(* PLC project Generated.project, CODESYS CODESYS V3.5 SP19 Patch 1 *)
(* stored: creationDateTime 2026-11-18T13:32:59.811305, modificationDateTime 2026-11-18T13:32:59.811305 *)

(* values of E_MachineHomingStep: IDLE: Referencement indisponible (Enable=FALSE); LOSS_SAFESTOP: Perte de datum en mouvement : arret controle en cours; BOTH_NOT_HOMED: Codeurs M1 et M2 non references : passer en MAINT_N2; M1_NOT_HOMED: Codeur M1 non reference ou mesure douteuse : homer M1; M2_NOT_HOMED: Codeur M2 non reference ou mesure douteuse : homer M2; OFFSET_UNKNOWN: Offset benne inconnu : passer en MAINT_N2; NEED_TOP_POSITION: Monter Both a vitesse lente jusqu au capteur haut; NEED_MECHANICAL_STOP: Capteur haut atteint : relacher la commande et attendre l arret; AWAIT_BUCKET_CONFIRM: Confirmer visuellement la benne : Fermee ou Ouverte; HOMING_IN_PROGRESS: Referencement conjoint M1/M2 en cours : ne pas manoeuvrer; VALID: Referencement machine valide : mode nominal disponible; FAILED: Referencement incomplet : rester en N2 et recommencer *)

{attribute 'qualified_only'}
{attribute 'strict'}
TYPE E_MachineHomingStep : (IDLE := 0, LOSS_SAFESTOP := 5, BOTH_NOT_HOMED := 10, M1_NOT_HOMED := 11, M2_NOT_HOMED := 12, OFFSET_UNKNOWN := 20, NEED_TOP_POSITION := 30, NEED_MECHANICAL_STOP := 40, AWAIT_BUCKET_CONFIRM := 45, HOMING_IN_PROGRESS := 50, VALID := 60, FAILED := 70);
END_TYPE

(* values of E_MachineHomingTxState: HX0_REPOS: Repos : N1 libre bloque si NOT Homed, M3 bloque N1/SEMI, attente 5s BP joy N1 ou BtnStart N2; HX1_BUCKET_PREPARE: M2 seul palier 1, ouv + ferm sans butees soft, garde continue 20s + decompte, BtnValidate neutre; HX2_CLIMB_TO_TOP: Couple M1+M2 palier 1 : montee lente + detente 2s max/geste, viser avant TOP sans toucher; HX3_TOP_CLEARANCE: Contact TOP = perdu/surcourse -> montee interdite, descente ~4s apres relachement TOP -> retour HX1; HX4_FINAL_CONFIRM: Arret avant TOP + avertissement -> BtnValidate neutre -> preset 8.5m M1+M2 + CommitClose -> Homed; HX7_FAILED: Echec / abandon : coupure mouvements, purge etats, attente Reset conscient *)

{attribute 'qualified_only'}
{attribute 'strict'}
TYPE E_MachineHomingTxState : (HX0_REPOS := 0, HX1_BUCKET_PREPARE := 1, HX2_CLIMB_TO_TOP := 2, HX3_TOP_CLEARANCE := 3, HX4_FINAL_CONFIRM := 4, HX7_FAILED := 5);
END_TYPE

(* values of E_Mode: DISABLE: Mode Désactivé / Veille de sécurité (sorties bloquées); MAINT_N1: Manuel Niveau 1 : Pilotage unitaire avec toutes sécurités actives; MAINT_N2: Manuel Niveau 2 : Pilotage dégradé (droits étendus + bypasses autorisés); SEMI_AUTO: Mode Semi-Automatique (séquenceur automatique) *)

{attribute 'qualified_only'}
{attribute 'strict'}
TYPE E_Mode : (DISABLE := 0, MAINT_N1 := 1, MAINT_N2 := 2, SEMI_AUTO := 3);
END_TYPE

(* ======================================================================= 🧩 ST_Fault — Brique socle défaut (2 vues : live + latchée) ─────────────────────────────────────────────────────────────── 🎯 Rôle : porter l'état défaut d'un composant, applicable dans TOUS les cas (acquittable ou non), sans brique warning séparée. • Vue LIVE (Error / ErrorId) : suit la cause, retombe seule à 0. • Vue LATCHÉE (Latched / LatchedId): mémorisée au défaut, reste jusqu'au front Reset. Le choix acquittable / non-acquittable se fait PAR CAUSE (ST_FaultCause.Latching), jamais par bloc. 🔒 Sécurité : interlock TOUJOURS sur la cause brute (Error / ErrorId), jamais sur l'acquittement. Reset TOUJOURS effectif, jamais conditionné (std §9). 🧬 Composition : brique de base réutilisable — sortie de FB, struct métier, GVL. Texte IHM NON stocké ici : dérivé côté IHM depuis LatchedId / ErrorId. 📄 Doc : DOC/STDS/CODE_QUALITY_STANDARDS.md §2quinquies / §9 ======================================================================= *)
TYPE ST_Fault : STRUCT
  Error : BOOL;  (* <-- [DIAG] vue LIVE : au moins une cause présente maintenant *)
  ErrorId : WORD;  (* <-- [DIAG] bitfield des causes présentes maintenant (0 si aucune) *)
  Latched : BOOL;  (* <-- [DIAG] vue LATCHÉE : défaut non acquitté, reste jusqu'au front Reset *)
  LatchedId : WORD;  (* <-- [DIAG] ErrorId figé à l'apparition du défaut, effacé au Reset *)
END_STRUCT;
END_TYPE

(* ======================================================================= 🧩 ST_FaultCause — Cause élémentaire alimentant ST_Fault (socle FB_FaultCore) ─────────────────────────────────────────────────────────────── 🎯 Rôle : une cause exprimée EN CLAIR (BOOL + libellé), sans bitfield ni masque. Le FB métier remplit une liste (ARRAY[0..15] OF ST_FaultCause) ; le socle FB_FaultCore en déduit ST_Fault (vue live + vue latchée). 🔒 Sécurité : interlock TOUJOURS sur Active (cause brute), jamais sur le latch. Latching = TRUE → la cause ARME la vue latchée (défaut à acquitter). Latching = FALSE → la cause n'alimente que la vue live (retombe seule). Fail-safe : une cause laissée à Latching=FALSE reste visible en live — pour la rendre acquittable, il faut le déclarer explicitement. 📄 Doc : DOC/STDS/CODE_QUALITY_STANDARDS.md §2quinquies / §9 ======================================================================= *)
TYPE ST_FaultCause : STRUCT
  Active : BOOL;  (* 1 = cause présente maintenant (interlock sur cette valeur) *)
  Latching : BOOL;  (* 1 = cause à acquitter (arme Latched) ; 0 = live seulement *)
  Texte : STRING;  (* libellé prêt IHM (non stocké dans ST_Fault, dérivé côté IHM) *)
END_STRUCT;
END_TYPE

(* ======================================================================= 🧩 ST_Lifecycle — Brique socle cycle d'exécution ─────────────────────────────────────────────────────────────── 🎯 Rôle : porter l'avancement d'une action à cycle (organe, séquenceur). Optionnelle : un FB purement synchrone (conditionneur, filtre, joystick) ne la porte pas. 🧬 Composition : brique de base réutilisable, composée avec ST_Fault. 📄 Doc : DOC/STDS/CODE_QUALITY_STANDARDS.md §2quinquies ======================================================================= *)
TYPE ST_Lifecycle : STRUCT
  Busy : BOOL;  (* <-- [STAT] 1 = action en cours *)
  Done : BOOL;  (* <-- [STAT] 1 = action terminée avec succès *)
END_STRUCT;
END_TYPE

(* ======================================================================= 🔌 ST_ProgramWinchRequest — Demande de mouvement treuil par le programme ─────────────────────────────────────────────────────────────── 🎯 Rôle : Regroupe les demandes logiques de treuil formulées par le séquenceur 📄 Référentiel : DOC/WFLOW/CONTRACTS/INTERPRG_CONTRACT_PRG03_MODES_CYCLE_v1.0.md ======================================================================= *)
TYPE ST_ProgramWinchRequest : STRUCT
  RunRequest : BOOL;  (* Ordre marche demandé par le programme *)
  ReqAscent : BOOL;  (* Demande montée *)
  ReqDescend : BOOL;  (* Demande descente *)
  StepTgt : INT;  (* Palier de vitesse cible demandé (1 à 5, 0 = arrêt) *)
END_STRUCT;
END_TYPE

(* ======================================================================= 🔌 ST_fbMachineHomingCycle_AxisHomingStatus — Statut homing d'un axe treuil ─────────────────────────────────────────────────────────────── 🎯 Rôle : Regroupe l'etat de homing d'un axe (M1 ou M2) consomme par FB_CycleMachineHoming pour piloter le guide et la transaction. 📄 Doc métier : DOC/AF/AF_Partie-09_Fonction_Encoder_v2.4.md (F09.08) ======================================================================= *)
TYPE ST_fbMachineHomingCycle_AxisHomingStatus : STRUCT
  HomedAndReliable : BOOL;  (* Codeur reference ET mesure jugee fiable (gate strict) *)
  HomingBusy : BOOL;  (* Sequence de homing en cours sur l'axe *)
  HomingDone : BOOL;  (* Homing termine avec succes (HomingLifecycle.Done cote FB_Encoder) *)
  HomingError : BOOL;  (* Homing en erreur sur l'axe (HomingFault.Error) *)
  HomingProvisional : BOOL;  (* TRUE si le datum persistant RETAIN est provisoire (HX1 0m) *)
END_STRUCT;
END_TYPE

(* ======================================================================= 🔌 ST_fbMachineHomingCycle_BucketCommit — Commit atomique de l'etat benne ─────────────────────────────────────────────────────────────── 🎯 Rôle : Impulsion 1 scan emise par FB_CycleMachineHoming vers FB_Bucket apres succes des DEUX homings. FB_Bucket reste seul proprietaire de IsOpen / IsClosed. 🔒 Sécurité : CommitOpen et CommitClose mutuellement exclusifs (garanti par le corps du FB — rejet du double-confirm, cf. C-2). 📄 Doc métier : DOC/AF/AF_Partie-05_Modes_Maintenance_v2.1.md ======================================================================= *)
TYPE ST_fbMachineHomingCycle_BucketCommit : STRUCT
  CommitOpen : BOOL;  (* Publier "benne ouverte" (impulsion 1 scan) *)
  CommitClose : BOOL;  (* Publier "benne fermee" (impulsion 1 scan) *)
  CommitInvalidate : BOOL;  (* Revoquer reference benne (abandon avant calibration altimetrie) *)
END_STRUCT;
END_TYPE

(* ======================================================================= ⚙️ ST_fbMachineHomingCycle_Cfg — Réglages de FB_CycleMachineHoming ─────────────────────────────────────────────────────────────────────── 🎯 Rôle : Réglages géométriques du référencement machine (cible haute M2/benne + écarts benne) + temporisations de garde du GRAFCET de homing (montée, homing axes). 🔒 Ownership : produit par PRG_02_Acquisition depuis _WinchM2CfgPersist (cible haute) et _BucketCfgPersist (écarts, GVL_PERSISTENT). Initialized : drapeau de restauration boot (pont persistant). 📄 Doc métier : DOC/AF/AF_Partie-09_Fonction_Encoder_v2.4.md (F09.08) ======================================================================= *)
TYPE ST_fbMachineHomingCycle_Cfg : STRUCT
  CfgTopHomingTarget_M : REAL;  (* Position capteur haut M2/benne (m) — cible finale HX4 M2 (+ OffsetCloseM) *)
  CfgTopHomingTargetM1_M : REAL := 8.5;  (* Position capteur haut M1 (m) — cible finale HX4 M1 (defaut 8.5 m) *)
  CfgOffsetOpen_M : REAL;  (* Ecart géométrique benne ouverte (m) *)
  CfgOffsetClose_M : REAL;  (* Ecart géométrique benne fermée (m) *)
  CfgTimeoutClimb : TIME := TIME#300s0ms;  (* Garde de montee : budget d'une MONTER CONTINUE (un temporisateur remet son temps ecoule a zero des que la commande retombe : une pause operateur ou un arret d'urgence ne consomme donc rien). Derivation : course maximale de cable = CfgTopSensorPos_M - CfgCableLimitDescent_M (8,5 m - (-50 m) = 58,5 m) ; borne haute de vitesse du palier 1 = 0,4 m/s (GVL_PERSISTENT._WinchSpeedConfig.SpeedBandMaxMps[1], valeur de banc A MESURER sur site) => 58,5 / 0,4 = 146,3 s ; marge x2 = 292,5 s ; valeur retenue 300 s (arrondie au-dessus). A revoir si la course ou la vitesse du palier 1 changent (gate G511). Garde de montee au capteur haut (0 = pas de garde) *)
  CfgEntryHoldTime : TIME := TIME#5s0ms;  (* Duree maintien BP joystick au neutre en HX0 (MAINT_N1) *)
  CfgBucketPrepareTimeout : TIME := TIME#20s0ms;  (* Duree max commande continue M2 en HX1 (coupe -> neutre) *)
  CfgSlackReliefMaxTime : TIME := TIME#2s0ms;  (* Duree max descente detente cable par geste en HX2 *)
  CfgTopClearanceTime : TIME := TIME#4s0ms;  (* Duree descente accumulee apres relachement TOP en HX3 *)
  CfgTimeoutHomeAxes : TIME := TIME#60s0ms;  (* Garde globale prise de reference (HX4) *)
  Initialized : BOOL := FALSE;  (* Drapeau de restauration config au boot (pont persistant) *)
END_STRUCT;
END_TYPE

(* ======================================================================= 🔌 ST_fbMachineHomingCycle_HomingDemand — Demande de homing conjoint vers un axe ─────────────────────────────────────────────────────────────── 🎯 Rôle : Ordre de prise d'origine emis par FB_CycleMachineHoming vers une facade FB_Encoder. M1 : cible configuree. M2 : cible geometrique dynamique (top M1 configure +/- offset benne), jamais une position M1 live. 📄 Doc métier : DOC/AF/AF_Partie-09_Fonction_Encoder_v2.4.md (F09.08) ======================================================================= *)
TYPE ST_fbMachineHomingCycle_HomingDemand : STRUCT
  HomeReq : BOOL;  (* Demande de prise d'origine pour cet axe (vocab reserve Homing) *)
  UseDynamicTarget : BOOL;  (* TRUE => cible = DynamicTarget_M (M2 uniquement) *)
  DynamicTarget_M : REAL;  (* Cible geometrique benne (m) : CfgTopHomingTargetM + offset *)
  Provisional : BOOL;  (* TRUE => marque Calib.HomingProvisional RETAIN (zero provisoire HX1) *)
END_STRUCT;
END_TYPE

(* ======================================================================= 🎯 FB_CycleMachineHoming — Cycle de referencement machine M1/M2/benne ─────────────────────────────────────────────────────────────── Role : GRAFCET sequentiel 5 etapes (HX0..HX4 + HX7_FAILED) : - HX0_REPOS : N1 libre bloque si NOT Homed, M3 verrouille N1/SEMI (echappatoire N2), entree par 5s BP joystick au neutre (N1) ou BtnStart (N2). Jamais relanceable si MachineHomed = TRUE. - HX1_BUCKET_PREPARE : M2 seul palier 1, ouv + ferm sans butees soft, garde continue 20s + decompte message, BtnValidate neutre. - HX2_CLIMB_TO_TOP : Couple M1+M2 palier 1, montee lente + detente cable max 2s par geste, viser avant TOP sans le toucher. - HX3_TOP_CLEARANCE : Contact TOP = surcourse/perdu -> coupure montee, descente ~4s accumulee apres relachement TOP -> retour HX1. - HX4_FINAL_CONFIRM : Arret avant TOP + avertissement + BtnValidate neutre -> preset 8.5m M1 + (8.5m + OffsetCloseM) M2 + CommitClose. Doc metier : DOC/WFLOW/MISE_EN_SERVICE/PLAN_REFONTE_GRAFCET_HOMING_20261118_v1.0.md + DOC/AF/AF_Partie-09_Fonction_Encoder_v2.4.md (F09.08) ======================================================================= *)
FUNCTION_BLOCK FB_CycleMachineHoming
  VAR_INPUT
    Enable : BOOL;  (* === CONTRAT STANDARD (Enable + Reset) === --> [CMD] Autorisation generale *)
    Reset : BOOL;  (* --> [CMD] Acquittement defaut / abandon cycle (front) *)
    Mode : E_Mode;  (* === MODE ARBITRE === --> [CMD] Mode machine (MAINT_N1 ou MAINT_N2 autorises) *)
    BootReady : BOOL;  (* --> [HW] Acquisition + codeurs valides apres boot *)
    TopPositionSensor : BOOL;  (* === PERMIS SECURITE === --> [SAFE] Capteur haut commun M1/M2 (TRUE = atteint) *)
    TopHardStopLatched : BOOL := FALSE;  (* --> [SAFE] Latch directionnel capteur haut (PRG_06_Outputs) *)
    WinchesMechanicallyStopped : BOOL;  (* --> [SAFE] M1 ET M2 arret mecanique confirme *)
    BucketIsOpen : BOOL := FALSE;  (* --> [HW] Benne ouverte confirmee (PRG_04_Treuils_Benne) *)
    M1Status : ST_fbMachineHomingCycle_AxisHomingStatus;  (* === ACQUISITION HOMING (M1 / M2) === --> [HW] Statut homing axe M1 *)
    M2Status : ST_fbMachineHomingCycle_AxisHomingStatus;  (* --> [HW] Statut homing axe M2 *)
    BucketOffsetValid : BOOL;  (* === ETAT BENNE === --> [HW] Reference benne persistante valide *)
    DeadmanArmed : BOOL;  (* === PERMIS OPERATEUR (joystick + homme-mort) === --> [CMD] Homme-mort arme *)
    RawDeadmanButton : BOOL := FALSE;  (* --> [HW] BP joystick brut (sert en HX0 N1 quand ArmingPermit=FALSE) *)
    JoystickDeflected : BOOL;  (* --> [CMD] Joystick deflechi (X ou Y hors neutre) *)
    JoystickPull : BOOL;  (* --> [CMD] Manche tire = montee / fermeture benne *)
    JoystickPush : BOOL;  (* --> [CMD] Manche pousse = descente / ouverture benne *)
    BtnValidation : BOOL;  (* === VALIDATION OPERATEUR === --> [CMD] Bouton validation IHM unifie (HX1, HX2->HX4, HX4) *)
    StartRequest : BOOL;  (* --> [CMD] Bouton Start IHM (HX0 en MAINT_N2) *)
    BtnConfirmHomingBucket : BOOL;  (* --> [CMD] Compat bouton IHM historique HX1 *)
    JoystickWinchSelectArbitrated : INT;  (* === INTERLOCK COUPLAGE E1 & RETOUR ARBITRAGE === --> [CMD] Selecteur treuil arbitre aval (0=couple, 2=M2) *)
    CablePosM1 : REAL;  (* === MESURES POSITIONS === --> [MEAS] Position cable M1 (m) *)
    CablePosM2 : REAL;  (* --> [MEAS] Position cable M2 (m) *)
    CoherenceLimitM : REAL := 1;  (* --> [CFG] Coherence (compat) *)
    CfgCommissioningEnable : BOOL;  (* === MISE EN SERVICE : forcage de step (encadre) === --> [CFG] Case mise en service *)
    CfgForceStepTarget : INT;  (* --> [CFG] Step cible [0..5] *)
    CfgForceStepApply : BOOL;  (* --> [CMD] Front d'application forcage *)
    Cfg : ST_fbMachineHomingCycle_Cfg;  (* === REGLAGES & CONFIGURATION === --> [CFG] Reglages + temporisations *)
  END_VAR
  VAR_OUTPUT
    Ready : BOOL;  (* === CONTRAT STANDARD === *)
    Fault : ST_Fault;
    Lifecycle : ST_Lifecycle;
    MachineHomed : BOOL;  (* === QUALIFICATION MACHINE === *)
    MachineHomingStep : E_MachineHomingStep := E_MachineHomingStep.IDLE;
    MachineHomingStepAtError : E_MachineHomingStep := E_MachineHomingStep.IDLE;
    MachineHomingSeqStep : E_MachineHomingTxState := E_MachineHomingTxState.HX0_REPOS;
    MachineHomingInstruction : STRING(120);
    MachineHomingActionText : STRING(120);
    MachineHomingActive : BOOL;
    MachineHomingLossSafeStop : BOOL;
    MachineHomingFailed : BOOL;
    HomingModeBActive : BOOL;
    M1Demand : ST_fbMachineHomingCycle_HomingDemand;  (* === DEMANDES HOMING (M1 / M2) === *)
    M2Demand : ST_fbMachineHomingCycle_HomingDemand;
    CmdWinchM1 : ST_ProgramWinchRequest;  (* === ORDRES / PERMIS VERS PRG_03 / PRG_04 === *)
    CmdWinchM2 : ST_ProgramWinchRequest;
    CmdBucketOpen : BOOL;
    CmdBucketClose : BOOL;
    CmdWinchSelect : INT := -1;
    AllowAscent : BOOL;
    AllowDescend : BOOL;
    SoftLimitsOff : BOOL;
    InvalidateProvisionalDatum : BOOL;
    BucketCommit : ST_fbMachineHomingCycle_BucketCommit;  (* === COMMIT BENNE === *)
    M3Locked : BOOL;  (* === VERROU TRANSLATION === *)
    TopContactLatched : BOOL;  (* === LATCH & COMPTEUR CONTACT TOP HOMING === *)
    TopContactCount : UINT;
  END_VAR
  VAR
    instFault : FB_FaultCore;  (* === SOUS-INSTANCES === *)
    ResetEdge : R_TRIG;
    LatchedEdge : R_TRIG;
    StartEdge : R_TRIG;
    BtnValidationEdge : R_TRIG;
    HomingBucketConfirmEdge : R_TRIG;
    ForceStepApplyEdge : R_TRIG;
    instCauses : ARRAY[0..15] OF ST_FaultCause;
    SeqStep : E_MachineHomingTxState := E_MachineHomingTxState.HX0_REPOS;  (* === GRAFCET & ETATS INTERNES === *)
    CommitPublished : BOOL;
    CycleRunning : BOOL;
    FirstScanDone : BOOL;
    RawBtnSeenReleased : BOOL;
    Step1MoveCutoff : BOOL;
    Step1PresetIssued : BOOL;
    Step2SlackCutoff : BOOL;
    Step3BucketOpenDone : BOOL;
    Step3ClearanceDone : BOOL;
    Step4PresetIssued : BOOL;
    Step4AutoConfirmPending : BOOL;
    ProvisionalDatumActive : BOOL;
    ProvisionalAborted : BOOL;
    ForceStepClamped : INT;
    EntryHoldTimer : TON;  (* === TEMPORISATIONS === *)
    RecoveryHoldTimer : TON;
    StepValidateHoldTimer : TON;
    Step1MoveTimer : TON;
    Step2SlackTimer : TON;
    Step3Timer : TON;
    Step3AccumTime : TIME;
    Step3SegTime : TIME;
    Step3RemainingTime : TIME;
    Step3TimerRunning : BOOL;
    ClimbTimer : TON;
    HomeAxesTimer : TON;
    CouplingSettleTimer : TON;
    CouplingViolationTimer : TON;
    SettleGraceTimer : TON;
    EntryRemSec : INT;  (* === CALCULS AFFICHAGE === *)
    RecoveryRemSec : INT;
    ValRemSec : INT;
    Step1RemSec : INT;
    Step3RemSec : INT;
    BothAxesHomed : BOOL;  (* === CONDITIONS INTERMEDIAIRES === *)
    CommitOrOffsetValid : BOOL;
    ClimbPermit : BOOL;
    TopBlockedAtEntry : BOOL;
    RecoveryCauseGone : BOOL;
    EffectiveResetPulse : BOOL;
    Step1MovingCmd : BOOL;
    Step2SlackCmd : BOOL;
    Step3DescendEngaged : BOOL;
    StepValidateAllowed : BOOL;
    StepValidateHoldActive : BOOL;
    IsInMovePhase : BOOL;
    AxisHomingError : BOOL;
    MotionOutOfPhase : BOOL;
    ModeChangedInCycle : BOOL;
    ClimbTimedOut : BOOL;
    HomeAxesTimedOut : BOOL;
    TransactionAbort : BOOL;
    ReHomingAckRequired : BOOL;
    MachineWasHomed : BOOL;
    HomingLossLatched : BOOL;
    MachineHomedRaw : BOOL;
    AxesDatumRaw : BOOL;
    PrevMode : E_Mode := E_Mode.DISABLE;  (* === CONTEXTE MODES & INTERLOCKS === *)
    ModeIsMaint1 : BOOL;
    ModeIsMaint2 : BOOL;
    MaintenanceActive : BOOL;
    ClimbStepActive : BOOL;
    ClimbCommandActive : BOOL;
    CouplingInterlockFault : BOOL;
    ValidatePressed : BOOL;
    CST_CauseHomingLostInMotion : INT := 0;
    CST_CauseClimbTimeout : INT := 1;
    CST_CauseMotionOutOfPhase : INT := 2;
    CST_CauseHomingErrorM1 : INT := 3;
    CST_CauseHomingErrorM2 : INT := 4;
    CST_CauseHomeAxesTimeout : INT := 5;
    CST_CauseCouplingFault : INT := 6;
    CST_SettleGrace : TIME := TIME#3s0ms;
  END_VAR

            

{region "§1 Fronts, remises a zero de tete de scan"}
IF NOT FirstScanDone THEN
    SeqStep              := E_MachineHomingTxState.HX0_REPOS;
    MachineHomingSeqStep := E_MachineHomingTxState.HX0_REPOS;
    MachineHomingFailed  := FALSE;
    HomingModeBActive    := FALSE;
    RawBtnSeenReleased   := NOT RawDeadmanButton;
    Step1MoveCutoff      := FALSE;
    Step1PresetIssued    := FALSE;
    Step2SlackCutoff     := FALSE;
    Step3BucketOpenDone  := FALSE;
    Step3ClearanceDone   := FALSE;
    Step3AccumTime       := T#0s;
    Step3SegTime         := T#0s;
    Step3RemainingTime   := T#0s;
    Step3TimerRunning    := FALSE;
    Step3Timer(IN := FALSE, PT := T#0s);
    EntryHoldTimer(IN := FALSE, PT := T#0s);
    RecoveryHoldTimer(IN := FALSE, PT := T#0s);
    StepValidateHoldTimer(IN := FALSE, PT := T#0s);
    Step4PresetIssued       := FALSE;
    Step4AutoConfirmPending := FALSE;
    ProvisionalDatumActive  := FALSE;
    ProvisionalAborted      := FALSE;
    TopContactLatched       := FALSE;
    TopContactCount         := 0;
    PrevMode                := Mode;
END_IF;

// Sorties impulsionnelles et permis remis a zero en tete de scan
M1Demand.HomeReq := FALSE; M1Demand.UseDynamicTarget := FALSE; M1Demand.DynamicTarget_M := 0.0; M1Demand.Provisional := FALSE;
M2Demand.HomeReq := FALSE; M2Demand.UseDynamicTarget := FALSE; M2Demand.DynamicTarget_M := 0.0; M2Demand.Provisional := FALSE;
BucketCommit.CommitOpen       := FALSE;
BucketCommit.CommitClose      := FALSE;
BucketCommit.CommitInvalidate := FALSE;
InvalidateProvisionalDatum    := FALSE;
CmdBucketOpen  := FALSE;
CmdBucketClose := FALSE;
CmdWinchM1.RunRequest := FALSE; CmdWinchM1.ReqAscent := FALSE; CmdWinchM1.ReqDescend := FALSE; CmdWinchM1.StepTgt := 0;
CmdWinchM2.RunRequest := FALSE; CmdWinchM2.ReqAscent := FALSE; CmdWinchM2.ReqDescend := FALSE; CmdWinchM2.StepTgt := 0;
CmdWinchSelect := -1;
AllowAscent    := FALSE;
AllowDescend   := FALSE;
SoftLimitsOff  := FALSE;

ResetEdge(CLK := Reset);
LatchedEdge(CLK := Fault.Latched);
StartEdge(CLK := StartRequest);
BtnValidationEdge(CLK := BtnValidation);
HomingBucketConfirmEdge(CLK := BtnConfirmHomingBucket);
ValidatePressed := BtnValidationEdge.Q OR HomingBucketConfirmEdge.Q;

ModeIsMaint1 := (Mode = E_Mode.MAINT_N1);
ModeIsMaint2 := (Mode = E_Mode.MAINT_N2);
MaintenanceActive := ModeIsMaint1 OR ModeIsMaint2;

CycleRunning  := (SeqStep <> E_MachineHomingTxState.HX0_REPOS);
IsInMovePhase := (SeqStep = E_MachineHomingTxState.HX1_BUCKET_PREPARE)
              OR (SeqStep = E_MachineHomingTxState.HX2_CLIMB_TO_TOP)
              OR (SeqStep = E_MachineHomingTxState.HX3_TOP_CLEARANCE);
{endregion}

{region "§2 Conditions intermediaires"}
BothAxesHomed       := M1Status.HomedAndReliable AND M2Status.HomedAndReliable;
CommitOrOffsetValid := CommitPublished OR BucketOffsetValid;
ClimbPermit         := DeadmanArmed AND JoystickPull AND NOT JoystickPush;

// Grace deceleration en HX4 / HX7
SettleGraceTimer(IN := (SeqStep = E_MachineHomingTxState.HX4_FINAL_CONFIRM)
                       OR (SeqStep = E_MachineHomingTxState.HX7_FAILED), PT := CST_SettleGrace);

AxisHomingError  := M1Status.HomingError OR M2Status.HomingError;
MotionOutOfPhase := CycleRunning AND NOT IsInMovePhase
                    AND NOT WinchesMechanicallyStopped AND SettleGraceTimer.Q;

// Garde de montee HX2 (consommee UNIQUEMENT pendant la montee commandee, gate G511)
ClimbStepActive    := (SeqStep = E_MachineHomingTxState.HX2_CLIMB_TO_TOP);
ClimbCommandActive := ClimbStepActive AND ClimbPermit;
ClimbTimer(IN := ClimbCommandActive, PT := Cfg.CfgTimeoutClimb);
ClimbTimedOut := ClimbStepActive AND (Cfg.CfgTimeoutClimb > T#0s) AND ClimbTimer.Q;
CouplingSettleTimer(IN := ClimbStepActive AND (JoystickWinchSelectArbitrated = 0), PT := T#300ms);

// Garde prise de reference provisoire HX1 (0m) et finale HX4 (8.5m)
HomeAxesTimer(
    IN := ((SeqStep = E_MachineHomingTxState.HX1_BUCKET_PREPARE) AND Step1PresetIssued)
          OR ((SeqStep = E_MachineHomingTxState.HX4_FINAL_CONFIRM) AND Step4PresetIssued
              AND NOT (M1Status.HomingDone AND M2Status.HomingDone AND NOT M1Status.HomingBusy AND NOT M2Status.HomingBusy)),
    PT := Cfg.CfgTimeoutHomeAxes
);
HomeAxesTimedOut := (((SeqStep = E_MachineHomingTxState.HX1_BUCKET_PREPARE) AND Step1PresetIssued)
                     OR ((SeqStep = E_MachineHomingTxState.HX4_FINAL_CONFIRM) AND Step4PresetIssued
                         AND NOT (M1Status.HomingDone AND M2Status.HomingDone AND NOT M1Status.HomingBusy AND NOT M2Status.HomingBusy)))
                    AND (Cfg.CfgTimeoutHomeAxes > T#0s)
                    AND HomeAxesTimer.Q;

// Violation couplage / selecteur (HX1 ou HX3A=M2 seul, HX2 ou HX3B=M1+M2 couple)
CouplingViolationTimer(
    IN := ((((SeqStep = E_MachineHomingTxState.HX2_CLIMB_TO_TOP)
             OR ((SeqStep = E_MachineHomingTxState.HX3_TOP_CLEARANCE) AND Step3BucketOpenDone))
            AND (JoystickWinchSelectArbitrated <> 0))
           OR (((SeqStep = E_MachineHomingTxState.HX1_BUCKET_PREPARE)
                OR ((SeqStep = E_MachineHomingTxState.HX3_TOP_CLEARANCE) AND NOT Step3BucketOpenDone))
               AND (JoystickWinchSelectArbitrated <> 2)))
          AND (JoystickPull OR JoystickPush),
    PT := T#600ms
);
CouplingInterlockFault := CouplingViolationTimer.Q;

TopBlockedAtEntry := TopPositionSensor OR TopHardStopLatched;
RecoveryCauseGone := BootReady AND NOT AxisHomingError AND NOT TopBlockedAtEntry AND NOT HomingLossLatched;
RecoveryHoldTimer(
    IN := Enable
          AND MaintenanceActive
          AND (SeqStep = E_MachineHomingTxState.HX7_FAILED)
          AND RecoveryCauseGone
          AND RawBtnSeenReleased
          AND RawDeadmanButton
          AND NOT JoystickDeflected
          AND WinchesMechanicallyStopped,
    PT := Cfg.CfgEntryHoldTime
);
EffectiveResetPulse := ResetEdge.Q OR RecoveryHoldTimer.Q;

// Changement de mode en cours de cycle (N1<->N2, DISABLE, SEMI_AUTO) : reset propre du graphe vers HX0
ModeChangedInCycle := FirstScanDone AND (Mode <> PrevMode)
                      AND (SeqStep <> E_MachineHomingTxState.HX0_REPOS)
                      AND (SeqStep <> E_MachineHomingTxState.HX7_FAILED);
TransactionAbort := CycleRunning
                    AND NOT ModeChangedInCycle
                    AND (AxisHomingError OR MotionOutOfPhase OR ClimbTimedOut
                         OR HomeAxesTimedOut OR CouplingInterlockFault);
{endregion}

{region "§3 Detection perte de datum"}
AxesDatumRaw    := BothAxesHomed;
MachineHomedRaw := AxesDatumRaw AND CommitOrOffsetValid AND NOT ProvisionalDatumActive
                   AND NOT ProvisionalAborted
                   AND NOT M1Status.HomingProvisional AND NOT M2Status.HomingProvisional
                   AND NOT ReHomingAckRequired;

IF FirstScanDone AND Enable AND NOT ProvisionalDatumActive AND NOT InvalidateProvisionalDatum
   AND NOT M1Status.HomingProvisional AND NOT M2Status.HomingProvisional
   AND NOT MachineHomedRaw AND MachineWasHomed THEN
    IF NOT WinchesMechanicallyStopped THEN
        HomingLossLatched := TRUE;
    END_IF;
    ReHomingAckRequired := TRUE;
END_IF;

IF Enable THEN
    MachineWasHomed := MachineHomedRaw;
END_IF;
MachineHomingLossSafeStop := HomingLossLatched AND NOT WinchesMechanicallyStopped;

IF EffectiveResetPulse AND WinchesMechanicallyStopped THEN
    HomingLossLatched   := FALSE;
    ReHomingAckRequired := FALSE;
END_IF;
{endregion}

{region "§4 Purge sur Reset & Forcage mise en service"}
IF EffectiveResetPulse OR ModeChangedInCycle
   OR ((SeqStep <> E_MachineHomingTxState.HX0_REPOS) AND (SeqStep <> E_MachineHomingTxState.HX7_FAILED) AND NOT MaintenanceActive) THEN
    IF ProvisionalDatumActive OR Step1PresetIssued OR M1Status.HomingProvisional OR M2Status.HomingProvisional THEN
        InvalidateProvisionalDatum    := TRUE;
        BucketCommit.CommitInvalidate := TRUE;
        ProvisionalDatumActive        := FALSE;
        ProvisionalAborted            := TRUE;
        CommitPublished               := FALSE;
    ELSIF EffectiveResetPulse THEN
        ProvisionalAborted            := FALSE;
    END_IF;
    IF EffectiveResetPulse THEN
        MachineHomingFailed := FALSE;
        TopContactLatched   := FALSE;
        TopContactCount     := 0;
    END_IF;
    HomingModeBActive       := FALSE;
    Step1MoveCutoff         := FALSE;
    Step1PresetIssued       := FALSE;
    Step2SlackCutoff        := FALSE;
    Step3BucketOpenDone     := FALSE;
    Step3ClearanceDone      := FALSE;
    Step3AccumTime          := T#0s;
    Step3SegTime            := T#0s;
    Step3RemainingTime      := T#0s;
    Step3TimerRunning       := FALSE;
    Step3Timer(IN := FALSE, PT := T#0s);
    StepValidateHoldTimer(IN := FALSE, PT := T#0s);
    Step4PresetIssued       := FALSE;
    Step4AutoConfirmPending := FALSE;
    RawBtnSeenReleased      := NOT RawDeadmanButton;
    SeqStep                 := E_MachineHomingTxState.HX0_REPOS;
    MachineHomingSeqStep    := E_MachineHomingTxState.HX0_REPOS;
END_IF;

ForceStepApplyEdge(CLK := CfgForceStepApply);
IF Enable AND CfgCommissioningEnable AND ModeIsMaint2 AND ForceStepApplyEdge.Q THEN
    ForceStepClamped := LIMIT(0, CfgForceStepTarget, 5);
    CASE ForceStepClamped OF
        0: SeqStep := E_MachineHomingTxState.HX0_REPOS;
        1: SeqStep := E_MachineHomingTxState.HX1_BUCKET_PREPARE;
        2: SeqStep := E_MachineHomingTxState.HX2_CLIMB_TO_TOP;
        3: SeqStep := E_MachineHomingTxState.HX3_TOP_CLEARANCE;
        4: SeqStep := E_MachineHomingTxState.HX4_FINAL_CONFIRM;
        5: SeqStep := E_MachineHomingTxState.HX7_FAILED;
    END_CASE;
    Step1MoveCutoff         := FALSE;
    Step2SlackCutoff        := FALSE;
    Step3BucketOpenDone     := (ForceStepClamped = 3) AND BucketIsOpen;
    Step3ClearanceDone      := FALSE;
    Step3AccumTime          := T#0s;
    Step3SegTime            := T#0s;
    Step3RemainingTime      := T#0s;
    Step3TimerRunning       := FALSE;
    Step3Timer(IN := FALSE, PT := T#0s);
    Step4PresetIssued       := FALSE;
    Step4AutoConfirmPending := FALSE;
    IF (ForceStepClamped <= 1) AND (ProvisionalDatumActive OR Step1PresetIssued OR M1Status.HomingProvisional OR M2Status.HomingProvisional) THEN
        InvalidateProvisionalDatum    := TRUE;
        BucketCommit.CommitInvalidate := TRUE;
        ProvisionalDatumActive        := FALSE;
        ProvisionalAborted            := (ForceStepClamped = 0);
        CommitPublished               := FALSE;
        Step1PresetIssued             := FALSE;
    END_IF;
    MachineHomingFailed := FALSE;
END_IF;
{endregion}

{region "§5 Table des causes & socle defaut"}
instCauses[CST_CauseHomingLostInMotion].Active   := HomingLossLatched OR ReHomingAckRequired;
instCauses[CST_CauseHomingLostInMotion].Latching := TRUE;
instCauses[CST_CauseHomingLostInMotion].Texte    := 'Perte de datum machine en mouvement : re-referencer';

instCauses[CST_CauseClimbTimeout].Active   := ClimbTimedOut;
instCauses[CST_CauseClimbTimeout].Latching := TRUE;
instCauses[CST_CauseClimbTimeout].Texte    := 'Montee au capteur haut non aboutie dans le temps imparti';

instCauses[CST_CauseMotionOutOfPhase].Active   := MotionOutOfPhase;
instCauses[CST_CauseMotionOutOfPhase].Latching := TRUE;
instCauses[CST_CauseMotionOutOfPhase].Texte    := 'Mouvement treuil detecte hors phase autorisee du cycle';

instCauses[CST_CauseHomingErrorM1].Active   := CycleRunning AND M1Status.HomingError;
instCauses[CST_CauseHomingErrorM1].Latching := TRUE;
instCauses[CST_CauseHomingErrorM1].Texte    := 'Erreur de homing codeur M1 pendant le referencement conjoint';

instCauses[CST_CauseHomingErrorM2].Active   := CycleRunning AND M2Status.HomingError;
instCauses[CST_CauseHomingErrorM2].Latching := TRUE;
instCauses[CST_CauseHomingErrorM2].Texte    := 'Erreur de homing codeur M2 pendant le referencement conjoint';

instCauses[CST_CauseHomeAxesTimeout].Active   := HomeAxesTimedOut;
instCauses[CST_CauseHomeAxesTimeout].Latching := TRUE;
instCauses[CST_CauseHomeAxesTimeout].Texte    := 'Prise de reference finale non obtenue dans le temps';

instCauses[CST_CauseCouplingFault].Active   := CouplingInterlockFault;
instCauses[CST_CauseCouplingFault].Latching := TRUE;
instCauses[CST_CauseCouplingFault].Texte    := 'Defaut de couplage treuils M1+M2 pendant referencement';

instFault(Enable := Enable, Reset := Reset OR RecoveryHoldTimer.Q, Causes := instCauses);
Fault := instFault.Fault;
{endregion}

{region "§7 Gate Enable"}
IF NOT Enable THEN
    M1Demand.HomeReq := FALSE; M1Demand.UseDynamicTarget := FALSE; M1Demand.DynamicTarget_M := 0.0; M1Demand.Provisional := FALSE;
    M2Demand.HomeReq := FALSE; M2Demand.UseDynamicTarget := FALSE; M2Demand.DynamicTarget_M := 0.0; M2Demand.Provisional := FALSE;
    BucketCommit.CommitOpen  := FALSE;
    BucketCommit.CommitClose := FALSE;
    IF ProvisionalDatumActive OR Step1PresetIssued OR InvalidateProvisionalDatum OR BucketCommit.CommitInvalidate THEN
        InvalidateProvisionalDatum    := TRUE;
        BucketCommit.CommitInvalidate := TRUE;
        ProvisionalDatumActive        := FALSE;
        ProvisionalAborted            := TRUE;
        CommitPublished               := FALSE;
    ELSE
        BucketCommit.CommitInvalidate := FALSE;
        InvalidateProvisionalDatum    := FALSE;
    END_IF;
    CmdBucketOpen  := FALSE;
    CmdBucketClose := FALSE;
    CmdWinchM1.RunRequest := FALSE; CmdWinchM1.ReqAscent := FALSE; CmdWinchM1.ReqDescend := FALSE; CmdWinchM1.StepTgt := 0;
    CmdWinchM2.RunRequest := FALSE; CmdWinchM2.ReqAscent := FALSE; CmdWinchM2.ReqDescend := FALSE; CmdWinchM2.StepTgt := 0;
    CmdWinchSelect := -1;
    AllowAscent    := FALSE;
    AllowDescend   := FALSE;
    SoftLimitsOff  := FALSE;
    Ready          := FALSE;
    Lifecycle.Busy := FALSE;
    Lifecycle.Done := FALSE;
    MachineHomingActive := FALSE;
    M3Locked       := FALSE;
    Step1MoveCutoff         := FALSE;
    Step1PresetIssued       := FALSE;
    Step2SlackCutoff        := FALSE;
    Step3BucketOpenDone     := FALSE;
    Step3ClearanceDone      := FALSE;
    Step3AccumTime          := T#0s;
    Step3SegTime            := T#0s;
    Step3RemainingTime      := T#0s;
    Step3TimerRunning       := FALSE;
    Step3Timer(IN := FALSE, PT := T#0s);
    EntryHoldTimer(IN := FALSE, PT := T#0s);
    RecoveryHoldTimer(IN := FALSE, PT := T#0s);
    StepValidateHoldTimer(IN := FALSE, PT := T#0s);
    Step4PresetIssued       := FALSE;
    Step4AutoConfirmPending := FALSE;
    SeqStep                 := E_MachineHomingTxState.HX0_REPOS;
    MachineHomingSeqStep    := E_MachineHomingTxState.HX0_REPOS;
    MachineHomingStep       := E_MachineHomingStep.IDLE;
    MachineHomingInstruction := 'Cycle homing desactive';
    MachineHomingActionText  := '';
    PrevMode                := Mode;
    RETURN;
END_IF;
{endregion}

{region "§8 GRAFCET de referencement machine (CASE SeqStep)"}
MachineHomedRaw := AxesDatumRaw AND CommitOrOffsetValid AND NOT ProvisionalDatumActive
                   AND NOT ProvisionalAborted
                   AND NOT M1Status.HomingProvisional AND NOT M2Status.HomingProvisional
                   AND NOT ReHomingAckRequired AND NOT MachineHomingFailed AND NOT Fault.Latched;

IF NOT RawDeadmanButton THEN
    RawBtnSeenReleased := TRUE;
END_IF;

StepValidateAllowed := ((SeqStep = E_MachineHomingTxState.HX1_BUCKET_PREPARE) AND NOT Step1MoveCutoff AND NOT Step1PresetIssued)
                    OR ((SeqStep = E_MachineHomingTxState.HX2_CLIMB_TO_TOP) AND CouplingSettleTimer.Q AND NOT TopBlockedAtEntry)
                    OR ((SeqStep = E_MachineHomingTxState.HX4_FINAL_CONFIRM) AND NOT Step4PresetIssued AND NOT TopBlockedAtEntry);
StepValidateHoldActive := Enable
                          AND MaintenanceActive
                          AND NOT Fault.Latched
                          AND NOT MachineHomingFailed
                          AND StepValidateAllowed
                          AND RawBtnSeenReleased
                          AND RawDeadmanButton
                          AND NOT JoystickDeflected
                          AND WinchesMechanicallyStopped;
StepValidateHoldTimer(IN := StepValidateHoldActive, PT := Cfg.CfgEntryHoldTime);
ValidatePressed := BtnValidationEdge.Q OR HomingBucketConfirmEdge.Q OR StepValidateHoldTimer.Q;

CASE SeqStep OF

    E_MachineHomingTxState.HX0_REPOS:
        CmdWinchSelect := -1;

        // Garde RETAIN post-coupure secteur (B1) : si les codeurs ont redemarre avec un
        // zero provisoire HX1 persistant (coupure/reset pendant HX2..HX4), purge immediate.
        IF M1Status.HomingProvisional OR M2Status.HomingProvisional THEN
            InvalidateProvisionalDatum    := TRUE;
            BucketCommit.CommitInvalidate := TRUE;
            ProvisionalAborted            := TRUE;
            CommitPublished               := FALSE;
        END_IF;

        EntryHoldTimer(
            IN := NOT MachineHomedRaw
                  AND BootReady
                  AND NOT Fault.Latched
                  AND NOT MachineHomingFailed
                  AND NOT TopBlockedAtEntry
                  AND MaintenanceActive
                  AND RawBtnSeenReleased
                  AND RawDeadmanButton
                  AND NOT JoystickDeflected
                  AND WinchesMechanicallyStopped,
            PT := Cfg.CfgEntryHoldTime
        );

        // Verrou absolu (D2) : impossible si machine deja referencee ou TOP non degage
        IF NOT MachineHomedRaw AND BootReady AND NOT Fault.Latched AND NOT MachineHomingFailed AND NOT TopBlockedAtEntry THEN
            IF (MaintenanceActive AND EntryHoldTimer.Q)
               OR (ModeIsMaint2 AND StartEdge.Q AND NOT JoystickDeflected AND WinchesMechanicallyStopped) THEN
                Step1MoveCutoff         := FALSE;
                Step1PresetIssued       := FALSE;
                Step2SlackCutoff        := FALSE;
                Step3BucketOpenDone     := FALSE;
                Step3ClearanceDone      := FALSE;
                Step3AccumTime          := T#0s;
                Step3SegTime            := T#0s;
                Step3RemainingTime      := T#0s;
                Step3TimerRunning       := FALSE;
                Step3Timer(IN := FALSE, PT := T#0s);
                Step4PresetIssued       := FALSE;
                Step4AutoConfirmPending := FALSE;
                ProvisionalDatumActive  := FALSE;
                ProvisionalAborted      := FALSE;
                RawBtnSeenReleased      := FALSE;
                SeqStep := E_MachineHomingTxState.HX1_BUCKET_PREPARE;
            END_IF;
        END_IF;

    E_MachineHomingTxState.HX1_BUCKET_PREPARE:
        // M2 seul palier 1, ouverture + fermeture autorisees sans aucune butee soft
        CmdWinchSelect := 2;
        SoftLimitsOff  := TRUE;

        IF Step1MoveCutoff AND NOT JoystickDeflected AND NOT DeadmanArmed AND NOT RawDeadmanButton THEN
            Step1MoveCutoff := FALSE;
        END_IF;

        Step1MovingCmd := NOT Step1PresetIssued
                          AND (JoystickWinchSelectArbitrated = 2)
                          AND DeadmanArmed
                          AND (JoystickPull XOR JoystickPush);
        Step1MoveTimer(IN := Step1MovingCmd AND NOT Step1MoveCutoff, PT := Cfg.CfgBucketPrepareTimeout);
        IF Step1MoveTimer.Q THEN
            Step1MoveCutoff := TRUE;
        END_IF;

        AllowAscent  := NOT Step1MoveCutoff AND NOT Step1PresetIssued;
        AllowDescend := NOT Step1MoveCutoff AND NOT Step1PresetIssued;

        IF TransactionAbort THEN
            IF ProvisionalDatumActive OR Step1PresetIssued THEN
                InvalidateProvisionalDatum    := TRUE;
                BucketCommit.CommitInvalidate := TRUE;
                ProvisionalDatumActive        := FALSE;
                ProvisionalAborted            := TRUE;
                CommitPublished               := FALSE;
            END_IF;
            Step1PresetIssued   := FALSE;
            MachineHomingFailed := TRUE;
            SeqStep := E_MachineHomingTxState.HX7_FAILED;
        ELSIF NOT Step1PresetIssued THEN
            IF ValidatePressed AND NOT JoystickDeflected AND WinchesMechanicallyStopped THEN
                // Zero provisoire codeurs (0m M1, 0m + OffsetCloseM M2) pour monter droit et connaitre etat benne
                M1Demand.HomeReq          := TRUE;
                M1Demand.UseDynamicTarget := TRUE;
                M1Demand.DynamicTarget_M  := 0.0;
                M1Demand.Provisional      := TRUE;
                M2Demand.HomeReq          := TRUE;
                M2Demand.UseDynamicTarget := TRUE;
                M2Demand.DynamicTarget_M  := Cfg.CfgOffsetClose_M;
                M2Demand.Provisional      := TRUE;
                Step1PresetIssued := TRUE;
            END_IF;
        ELSIF BothAxesHomed AND M1Status.HomingDone AND M2Status.HomingDone
              AND NOT M1Status.HomingBusy AND NOT M2Status.HomingBusy THEN
            BucketCommit.CommitClose := TRUE;
            CommitPublished          := FALSE;
            ProvisionalDatumActive   := TRUE;
            ProvisionalAborted       := FALSE;
            Step1PresetIssued        := FALSE;
            Step2SlackCutoff         := FALSE;
            RawBtnSeenReleased       := FALSE;
            SeqStep := E_MachineHomingTxState.HX2_CLIMB_TO_TOP;
        END_IF;

    E_MachineHomingTxState.HX2_CLIMB_TO_TOP:
        // Couple M1+M2 palier 1 : montee lente + detente cable 2s max par geste.
        // Toucher TopPositionSensor = PERDU / surcourse -> coupure montee et Step 3.
        CmdWinchSelect := 0;
        SoftLimitsOff  := TRUE;

        IF Step2SlackCutoff AND NOT JoystickDeflected THEN
            Step2SlackCutoff := FALSE;
        END_IF;

        Step2SlackCmd := CouplingSettleTimer.Q
                         AND DeadmanArmed
                         AND JoystickPush AND NOT JoystickPull;
        Step2SlackTimer(IN := Step2SlackCmd AND NOT Step2SlackCutoff, PT := Cfg.CfgSlackReliefMaxTime);
        IF Step2SlackTimer.Q THEN
            Step2SlackCutoff := TRUE;
        END_IF;

        AllowAscent  := CouplingSettleTimer.Q AND NOT TopBlockedAtEntry;
        AllowDescend := CouplingSettleTimer.Q AND NOT Step2SlackCutoff;

        IF TransactionAbort THEN
            IF ProvisionalDatumActive THEN
                InvalidateProvisionalDatum    := TRUE;
                BucketCommit.CommitInvalidate := TRUE;
                ProvisionalDatumActive        := FALSE;
                ProvisionalAborted            := TRUE;
                CommitPublished               := FALSE;
            END_IF;
            MachineHomingFailed := TRUE;
            SeqStep := E_MachineHomingTxState.HX7_FAILED;
        ELSIF TopBlockedAtEntry THEN
            TopContactLatched   := TRUE;
            TopContactCount     := TopContactCount + UINT#1;
            AllowAscent         := FALSE;
            Step3BucketOpenDone := BucketIsOpen;
            Step3ClearanceDone  := FALSE;
            Step3AccumTime      := T#0s;
            Step3SegTime        := T#0s;
            Step3RemainingTime  := Cfg.CfgTopClearanceTime;
            Step3TimerRunning   := FALSE;
            Step3Timer(IN := FALSE, PT := T#0s);
            SeqStep := E_MachineHomingTxState.HX3_TOP_CLEARANCE;
        ELSIF ValidatePressed AND CouplingSettleTimer.Q AND NOT JoystickDeflected
              AND WinchesMechanicallyStopped AND NOT TopBlockedAtEntry THEN
            Step4PresetIssued       := FALSE;
            Step4AutoConfirmPending := TRUE;
            RawBtnSeenReleased      := NOT RawDeadmanButton;
            SeqStep := E_MachineHomingTxState.HX4_FINAL_CONFIRM;
        END_IF;

    E_MachineHomingTxState.HX3_TOP_CLEARANCE:
        // Contact TOP touche : 1) ouvrir benne prudemment (M2 seul, si pas deja ouverte),
        // puis 2) descente couplee M1+M2 accumulee ~4s apres capteur libre -> retour HX1.
        SoftLimitsOff := TRUE;
        AllowAscent   := FALSE;

        IF NOT Step3BucketOpenDone AND BucketIsOpen AND NOT JoystickDeflected AND WinchesMechanicallyStopped THEN
            Step3BucketOpenDone := TRUE;
        END_IF;

        IF NOT Step3BucketOpenDone THEN
            CmdWinchSelect := 2;
            AllowDescend   := TRUE;
            Step3TimerRunning := FALSE;
            Step3Timer(IN := FALSE, PT := T#0s);
        ELSE
            CmdWinchSelect := 0;

            IF TopPositionSensor THEN
                Step3AccumTime     := T#0s;
                Step3SegTime       := T#0s;
                Step3RemainingTime := Cfg.CfgTopClearanceTime;
                Step3ClearanceDone := FALSE;
                Step3TimerRunning  := FALSE;
                Step3Timer(IN := FALSE, PT := T#0s);
            ELSE
                Step3DescendEngaged := NOT Step3ClearanceDone
                                       AND (JoystickWinchSelectArbitrated = 0)
                                       AND DeadmanArmed
                                       AND JoystickPush AND NOT JoystickPull;

                IF Step3DescendEngaged THEN
                    IF NOT Step3TimerRunning THEN
                        IF Step3AccumTime >= Cfg.CfgTopClearanceTime THEN
                            Step3RemainingTime := T#0s;
                            Step3ClearanceDone := TRUE;
                        ELSE
                            Step3RemainingTime := Cfg.CfgTopClearanceTime - Step3AccumTime;
                        END_IF;
                        Step3Timer(IN := FALSE, PT := T#0s);
                        Step3TimerRunning := NOT Step3ClearanceDone;
                    END_IF;
                    IF Step3TimerRunning THEN
                        Step3Timer(IN := TRUE, PT := Step3RemainingTime);
                        Step3SegTime := Step3Timer.ET;
                        IF Step3Timer.Q THEN
                            Step3ClearanceDone := TRUE;
                            Step3AccumTime     := Cfg.CfgTopClearanceTime;
                            Step3SegTime       := T#0s;
                            Step3TimerRunning  := FALSE;
                            Step3Timer(IN := FALSE, PT := T#0s);
                        END_IF;
                    END_IF;
                ELSE
                    IF Step3TimerRunning THEN
                        Step3Timer(IN := TRUE, PT := Step3RemainingTime);
                        Step3AccumTime := Step3AccumTime + Step3Timer.ET;
                        IF Step3AccumTime >= Cfg.CfgTopClearanceTime THEN
                            Step3AccumTime     := Cfg.CfgTopClearanceTime;
                            Step3ClearanceDone := TRUE;
                        END_IF;
                        Step3SegTime      := T#0s;
                        Step3TimerRunning := FALSE;
                        Step3Timer(IN := FALSE, PT := T#0s);
                    END_IF;
                    IF Step3AccumTime >= Cfg.CfgTopClearanceTime THEN
                        Step3RemainingTime := T#0s;
                    ELSE
                        Step3RemainingTime := Cfg.CfgTopClearanceTime - Step3AccumTime;
                    END_IF;
                END_IF;
            END_IF;

            AllowDescend := NOT Step3ClearanceDone;
        END_IF;

        IF TransactionAbort THEN
            IF ProvisionalDatumActive THEN
                InvalidateProvisionalDatum    := TRUE;
                BucketCommit.CommitInvalidate := TRUE;
                ProvisionalDatumActive        := FALSE;
                ProvisionalAborted            := TRUE;
                CommitPublished               := FALSE;
            END_IF;
            Step3BucketOpenDone := FALSE;
            MachineHomingFailed := TRUE;
            SeqStep := E_MachineHomingTxState.HX7_FAILED;
        ELSIF Step3BucketOpenDone AND Step3ClearanceDone AND NOT TopPositionSensor AND NOT JoystickDeflected AND WinchesMechanicallyStopped THEN
            TopContactLatched   := FALSE;
            Step1MoveCutoff     := FALSE;
            Step3BucketOpenDone := FALSE;
            RawBtnSeenReleased  := NOT RawDeadmanButton;
            SeqStep := E_MachineHomingTxState.HX1_BUCKET_PREPARE;
        END_IF;

    E_MachineHomingTxState.HX4_FINAL_CONFIRM:
        // Zero mouvement : validation unique heritee de HX2 (ou explicite en forcage step 4)
        // -> ecriture 8.5m M1 + (8.5m + OffsetCloseM) M2 + CommitClose
        CmdWinchSelect := 0;
        SoftLimitsOff  := FALSE;
        AllowAscent    := FALSE;
        AllowDescend   := FALSE;

        IF TransactionAbort THEN
            IF ProvisionalDatumActive THEN
                InvalidateProvisionalDatum    := TRUE;
                BucketCommit.CommitInvalidate := TRUE;
                ProvisionalDatumActive        := FALSE;
                ProvisionalAborted            := TRUE;
                CommitPublished               := FALSE;
            END_IF;
            Step4PresetIssued       := FALSE;
            Step4AutoConfirmPending := FALSE;
            MachineHomingFailed     := TRUE;
            SeqStep := E_MachineHomingTxState.HX7_FAILED;
        ELSIF TopBlockedAtEntry THEN
            // Surcourse detectee pendant l'attente -> repli degagement Step 3, annule preset HX4 si arme
            TopContactLatched  := TRUE;
            TopContactCount    := TopContactCount + UINT#1;
            IF Step4PresetIssued THEN
                InvalidateProvisionalDatum    := TRUE;
                BucketCommit.CommitInvalidate := TRUE;
                ProvisionalDatumActive        := FALSE;
                ProvisionalAborted            := TRUE;
                CommitPublished               := FALSE;
            END_IF;
            Step4PresetIssued       := FALSE;
            Step4AutoConfirmPending := FALSE;
            Step3BucketOpenDone     := BucketIsOpen;
            Step3ClearanceDone      := FALSE;
            Step3AccumTime          := T#0s;
            Step3SegTime            := T#0s;
            Step3RemainingTime      := Cfg.CfgTopClearanceTime;
            Step3TimerRunning       := FALSE;
            Step3Timer(IN := FALSE, PT := T#0s);
            SeqStep := E_MachineHomingTxState.HX3_TOP_CLEARANCE;
        ELSIF NOT Step4PresetIssued THEN
            IF (Step4AutoConfirmPending OR ValidatePressed) AND NOT JoystickDeflected AND WinchesMechanicallyStopped THEN
                Step4AutoConfirmPending   := FALSE;
                M1Demand.HomeReq          := TRUE;
                M1Demand.UseDynamicTarget := TRUE;
                M1Demand.DynamicTarget_M  := Cfg.CfgTopHomingTargetM1_M;
                M2Demand.HomeReq          := TRUE;
                M2Demand.UseDynamicTarget := TRUE;
                M2Demand.DynamicTarget_M  := Cfg.CfgTopHomingTarget_M + Cfg.CfgOffsetClose_M;
                Step4PresetIssued := TRUE;
            END_IF;
        ELSIF BothAxesHomed AND M1Status.HomingDone AND M2Status.HomingDone
              AND NOT M1Status.HomingBusy AND NOT M2Status.HomingBusy AND NOT TopBlockedAtEntry THEN
            BucketCommit.CommitClose := TRUE;
            CommitPublished          := TRUE;
            ProvisionalDatumActive   := FALSE;
            ProvisionalAborted       := FALSE;
            ReHomingAckRequired      := FALSE;
            Step4PresetIssued        := FALSE;
            Step4AutoConfirmPending  := FALSE;
            RawBtnSeenReleased       := NOT RawDeadmanButton;
            SeqStep := E_MachineHomingTxState.HX0_REPOS;
        END_IF;

    E_MachineHomingTxState.HX7_FAILED:
        CmdWinchSelect := -1;
        SoftLimitsOff  := FALSE;
        AllowAscent    := FALSE;
        AllowDescend   := FALSE;

    ELSE
        MachineHomingFailed := TRUE;
        SeqStep := E_MachineHomingTxState.HX7_FAILED;

END_CASE;
{endregion}

{region "§9 Cycle de vie & qualification de sortie"}
CycleRunning := (SeqStep <> E_MachineHomingTxState.HX0_REPOS);

IF (SeqStep = E_MachineHomingTxState.HX1_BUCKET_PREPARE) THEN
    CmdWinchSelect := 2;
    SoftLimitsOff  := TRUE;
    AllowAscent    := NOT Step1MoveCutoff AND NOT Step1PresetIssued;
    AllowDescend   := NOT Step1MoveCutoff AND NOT Step1PresetIssued;
ELSIF (SeqStep = E_MachineHomingTxState.HX2_CLIMB_TO_TOP) THEN
    CmdWinchSelect := 0;
    SoftLimitsOff  := TRUE;
    AllowAscent    := CouplingSettleTimer.Q AND NOT TopBlockedAtEntry;
    AllowDescend   := CouplingSettleTimer.Q AND NOT Step2SlackCutoff;
ELSIF (SeqStep = E_MachineHomingTxState.HX3_TOP_CLEARANCE) THEN
    IF NOT Step3BucketOpenDone THEN
        CmdWinchSelect := 2;
        AllowDescend   := TRUE;
    ELSE
        CmdWinchSelect := 0;
        AllowDescend   := NOT Step3ClearanceDone;
    END_IF;
    SoftLimitsOff  := TRUE;
    AllowAscent    := FALSE;
ELSIF (SeqStep = E_MachineHomingTxState.HX4_FINAL_CONFIRM) THEN
    CmdWinchSelect := 0;
    SoftLimitsOff  := FALSE;
    AllowAscent    := FALSE;
    AllowDescend   := FALSE;
ELSE
    CmdWinchSelect := -1;
    SoftLimitsOff  := FALSE;
    AllowAscent    := FALSE;
    AllowDescend   := FALSE;
END_IF;

CommitOrOffsetValid := CommitPublished OR BucketOffsetValid;
MachineHomed := BothAxesHomed AND CommitOrOffsetValid
                AND NOT ProvisionalDatumActive
                AND NOT ProvisionalAborted
                AND NOT M1Status.HomingProvisional AND NOT M2Status.HomingProvisional
                AND (SeqStep <> E_MachineHomingTxState.HX7_FAILED)
                AND NOT MachineHomingFailed AND NOT ReHomingAckRequired
                AND NOT Fault.Latched;

// M3 verrouille des Step 0 en N1/SEMI si non reference (echappatoire N2 preservee en Step 0)
M3Locked             := CycleRunning OR (NOT MachineHomed AND NOT ModeIsMaint2);
MachineHomingActive  := (SeqStep = E_MachineHomingTxState.HX1_BUCKET_PREPARE)
                     OR (SeqStep = E_MachineHomingTxState.HX2_CLIMB_TO_TOP)
                     OR (SeqStep = E_MachineHomingTxState.HX3_TOP_CLEARANCE)
                     OR (SeqStep = E_MachineHomingTxState.HX4_FINAL_CONFIRM);
Lifecycle.Busy       := MachineHomingActive;
Lifecycle.Done       := CommitPublished AND (SeqStep = E_MachineHomingTxState.HX0_REPOS);
MachineHomingSeqStep := SeqStep;
{endregion}

{region "§10 Guide operateur — messages ASCII sans accents"}
IF Fault.Latched OR MachineHomingFailed OR (SeqStep = E_MachineHomingTxState.HX7_FAILED) THEN
    MachineHomingStep := E_MachineHomingStep.FAILED;
    IF RecoveryHoldTimer.ET > T#0s THEN
        RecoveryRemSec := DINT_TO_INT((TIME_TO_DINT(Cfg.CfgEntryHoldTime - RecoveryHoldTimer.ET) + DINT#999) / DINT#1000);
        IF RecoveryRemSec < 0 THEN RecoveryRemSec := 0; END_IF;
        MachineHomingInstruction := CONCAT('HX7 - Acquittement homing: ',
                                           CONCAT(INT_TO_STRING(RecoveryRemSec), 's'));
        MachineHomingActionText  := CONCAT('[HOMING] RELACHER=ANNULER - Acquitter dans ',
                                           CONCAT(INT_TO_STRING(RecoveryRemSec), 's'));
    ELSIF TopBlockedAtEntry THEN
        MachineHomingInstruction := 'HX7 - CAPTEUR TOP NON DEGAGE - Echec homing';
        IF ModeIsMaint2 THEN
            MachineHomingActionText := '[TREUIL] DESCENDRE pour degager capteur TOP puis Reset';
        ELSE
            MachineHomingActionText := '[SECURITE] TOP NON DEGAGE - Passer N2 pour descendre + Reset';
        END_IF;
    ELSIF RecoveryCauseGone THEN
        MachineHomingInstruction := 'HX7 - Echec homing - Tenir homme-mort 5s neutre (ou Reset)';
        MachineHomingActionText  := '[HOMING] Echec - Relacher puis HOMME-MORT 5s NEUTRE (ou Reset)';
    ELSE
        MachineHomingInstruction := 'HX7 - Defaut codeur actif - Verifier puis Reset';
        MachineHomingActionText  := '[HOMING] Defaut actif - Attendre retour codeurs puis Reset';
    END_IF;
ELSIF MachineHomingLossSafeStop THEN
    MachineHomingStep := E_MachineHomingStep.LOSS_SAFESTOP;
    MachineHomingInstruction := 'Reference perdue - Arret controle';
    MachineHomingActionText  := '[SECURITE] Reference perdue en mouvement - Acquitter (Reset)';
ELSIF MachineHomed AND NOT CycleRunning THEN
    MachineHomingStep := E_MachineHomingStep.VALID;
    MachineHomingInstruction := 'Homing fait';
    MachineHomingActionText  := '';
ELSIF (SeqStep = E_MachineHomingTxState.HX1_BUCKET_PREPARE) THEN
    MachineHomingStep := E_MachineHomingStep.AWAIT_BUCKET_CONFIRM;
    IF Step1PresetIssued THEN
        MachineHomingInstruction := 'HX1 - Prise 0m codeurs + benne fermee...';
        MachineHomingActionText  := '[HOMING] Enregistrement reference 0m + benne fermee...';
    ELSIF Step1MoveCutoff THEN
        MachineHomingInstruction := 'HX1 - DELAI 20s ATTEINT: relacher neutre et homme-mort';
        MachineHomingActionText  := '[HOMING] RELACHER joystick au neutre et homme-mort pour continuer';
    ELSIF StepValidateHoldActive THEN
        ValRemSec := DINT_TO_INT((TIME_TO_DINT(Cfg.CfgEntryHoldTime - StepValidateHoldTimer.ET) + DINT#999) / DINT#1000);
        IF ValRemSec < 0 THEN ValRemSec := 0; END_IF;
        MachineHomingInstruction := CONCAT('HX1 - CONFIRMATION BENNE FERMEE (0m): ',
                                           CONCAT(INT_TO_STRING(ValRemSec), 's'));
        MachineHomingActionText  := CONCAT('[BENNE] Tenir HOMME-MORT neutre: ',
                                           CONCAT(INT_TO_STRING(ValRemSec), 's = VALIDER FERMEE'));
    ELSE
        Step1RemSec := DINT_TO_INT((TIME_TO_DINT(Cfg.CfgBucketPrepareTimeout - Step1MoveTimer.ET) + DINT#999) / DINT#1000);
        IF Step1RemSec < 0 THEN Step1RemSec := 0; END_IF;
        MachineHomingInstruction := CONCAT('HX1 - FERMER BENNE M2 ',
                                           CONCAT(INT_TO_STRING(Step1RemSec), 's (AUCUNE BUTEE!)'));
        MachineHomingActionText  := '[BENNE] FERMER PRUDEMMENT (SANS BUTEES) puis HOMME-MORT 5s NEUTRE = 0m';
    END_IF;
ELSIF (SeqStep = E_MachineHomingTxState.HX2_CLIMB_TO_TOP) THEN
    MachineHomingStep := E_MachineHomingStep.NEED_TOP_POSITION;
    IF Step2SlackCutoff THEN
        MachineHomingInstruction := 'HX2 - Detente 2s atteinte: relacher neutre';
        MachineHomingActionText  := '[TREUIL] RELACHER joystick au neutre pour rearmer descente';
    ELSIF TopContactLatched AND TopBlockedAtEntry THEN
        MachineHomingInstruction := 'HX2 - Refus montee: contact TOP encore actif';
        MachineHomingActionText  := '[SECURITE] TOP actif - OUVRIR benne puis plonger pour degager';
    ELSIF StepValidateHoldActive THEN
        ValRemSec := DINT_TO_INT((TIME_TO_DINT(Cfg.CfgEntryHoldTime - StepValidateHoldTimer.ET) + DINT#999) / DINT#1000);
        IF ValRemSec < 0 THEN ValRemSec := 0; END_IF;
        MachineHomingInstruction := CONCAT('HX2 - CALIBRATION FINALE 8.5m: ',
                                           CONCAT(INT_TO_STRING(ValRemSec), 's'));
        MachineHomingActionText  := CONCAT('[HOMING] Tenir HOMME-MORT neutre: ',
                                           CONCAT(INT_TO_STRING(ValRemSec), 's = VALIDER 8.5m'));
    ELSIF TopContactCount > 0 THEN
        MachineHomingInstruction := CONCAT('HX2 - Approche plus basse (TOP:',
                                           CONCAT(UINT_TO_STRING(TopContactCount), ')'));
        MachineHomingActionText  := '[TREUIL] MONTER SOUS TOP (NE PAS TOUCHER) puis HOMME-MORT 5s NEUTRE';
    ELSE
        MachineHomingInstruction := 'HX2 - MONTER LENTEMENT SOUS CAPTEUR TOP (AUCUNE BUTEE)';
        MachineHomingActionText  := '[TREUIL] MONTER SOUS TOP sans le toucher puis HOMME-MORT 5s NEUTRE';
    END_IF;
ELSIF (SeqStep = E_MachineHomingTxState.HX3_TOP_CLEARANCE) THEN
    MachineHomingStep := E_MachineHomingStep.HOMING_IN_PROGRESS;
    IF NOT Step3BucketOpenDone THEN
        IF BucketIsOpen THEN
            MachineHomingInstruction := 'HX3 - Benne ouverte: relacher neutre pour plonger';
            MachineHomingActionText  := '[BENNE] BENNE OUVERTE - Relacher joystick au neutre pour plonger';
        ELSE
            MachineHomingInstruction := 'HX3 - TOP touche: OUVRIR BENNE PRUDEMMENT (M2 seul)';
            MachineHomingActionText  := '[BENNE] OUVRIR BENNE PRUDEMMENT (M2 seul) avant plongee degagement';
        END_IF;
    ELSIF TopPositionSensor THEN
        MachineHomingInstruction := 'HX3 - TOP touche: plonger/descendre couple pour degager';
        MachineHomingActionText  := '[TREUIL] PLONGER / DESCENDRE COUPLE pour degager capteur TOP';
    ELSIF Step3ClearanceDone THEN
        MachineHomingInstruction := 'HX3 - Degagement OK, relacher neutre -> retour HX1';
        MachineHomingActionText  := '[TREUIL] RELACHER joystick au neutre -> retour fermeture benne';
    ELSE
        Step3RemSec := DINT_TO_INT((TIME_TO_DINT(Step3RemainingTime - Step3SegTime) + DINT#999) / DINT#1000);
        IF Step3RemSec < 0 THEN Step3RemSec := 0; END_IF;
        MachineHomingInstruction := CONCAT('HX3 - Continuer descente degagement: ',
                                           CONCAT(INT_TO_STRING(Step3RemSec), 's'));
        MachineHomingActionText  := CONCAT('[TREUIL] DESCENDRE pour degager TOP: ',
                                           CONCAT(INT_TO_STRING(Step3RemSec), 's'));
    END_IF;
ELSIF (SeqStep = E_MachineHomingTxState.HX4_FINAL_CONFIRM) THEN
    MachineHomingStep := E_MachineHomingStep.AWAIT_BUCKET_CONFIRM;
    IF Step4PresetIssued OR Step4AutoConfirmPending THEN
        MachineHomingInstruction := 'HX4 - Ecriture references 8.5m + benne...';
        MachineHomingActionText  := '[HOMING] Calibration 8.5m + benne fermee en cours...';
    ELSIF StepValidateHoldActive THEN
        ValRemSec := DINT_TO_INT((TIME_TO_DINT(Cfg.CfgEntryHoldTime - StepValidateHoldTimer.ET) + DINT#999) / DINT#1000);
        IF ValRemSec < 0 THEN ValRemSec := 0; END_IF;
        MachineHomingInstruction := CONCAT('HX4 - Calibrer 8.5m + benne: ',
                                           CONCAT(INT_TO_STRING(ValRemSec), 's'));
        MachineHomingActionText  := CONCAT('[HOMING] Tenir HOMME-MORT neutre: ',
                                           CONCAT(INT_TO_STRING(ValRemSec), 's'));
    ELSE
        MachineHomingInstruction := 'HX4 - Calibrer 8.5m + benne? Homme-mort 5s neutre';
        MachineHomingActionText  := '[HOMING] Tenir HOMME-MORT 5s NEUTRE = calibrer 8.5m';
    END_IF;
ELSIF TopBlockedAtEntry THEN
    MachineHomingStep := E_MachineHomingStep.BOTH_NOT_HOMED;
    IF ModeIsMaint2 THEN
        MachineHomingInstruction := 'HX0 - CAPTEUR TOP NON DEGAGE (homing bloque)';
        MachineHomingActionText  := '[TREUIL] DESCENDRE pour degager capteur TOP puis Reset';
    ELSIF ModeIsMaint1 THEN
        MachineHomingInstruction := 'HX0 - CAPTEUR TOP NON DEGAGE (homing bloque)';
        MachineHomingActionText  := '[SECURITE] TOP NON DEGAGE - Passer N2 pour descendre + Reset';
    ELSE
        MachineHomingInstruction := 'HX0 - CAPTEUR TOP NON DEGAGE - Passer N2';
        MachineHomingActionText  := '[SECURITE] TOP NON DEGAGE - Passer N2 pour descendre';
    END_IF;
ELSIF ModeIsMaint1 THEN
    MachineHomingStep := E_MachineHomingStep.BOTH_NOT_HOMED;
    IF NOT BootReady THEN
        MachineHomingInstruction := 'HX0 - Attente prets codeurs/boot...';
        MachineHomingActionText  := '[HOMING] Attente codeurs prets...';
    ELSIF EntryHoldTimer.ET >= T#1500ms THEN
        EntryRemSec := DINT_TO_INT((TIME_TO_DINT(Cfg.CfgEntryHoldTime - EntryHoldTimer.ET) + DINT#999) / DINT#1000);
        IF EntryRemSec < 0 THEN EntryRemSec := 0; END_IF;
        MachineHomingInstruction := CONCAT('HX0 - LANCEMENT HOMING DANS ',
                                           CONCAT(INT_TO_STRING(EntryRemSec), 's (lacher=annul.)'));
        MachineHomingActionText  := CONCAT('[HOMING] LANCEMENT DANS ',
                                           CONCAT(INT_TO_STRING(EntryRemSec), 's - LACHER POUR ANNULER'));
    ELSIF ProvisionalAborted AND NOT RawDeadmanButton THEN
        MachineHomingInstruction := 'HX0 - Altimetrie non calibree: re-referencer';
        MachineHomingActionText  := '[HOMING] Tenir HOMME-MORT 5s NEUTRE pour relancer';
    ELSIF RawDeadmanButton AND NOT JoystickDeflected AND RawBtnSeenReleased THEN
        EntryRemSec := DINT_TO_INT((TIME_TO_DINT(Cfg.CfgEntryHoldTime - EntryHoldTimer.ET) + DINT#999) / DINT#1000);
        IF EntryRemSec < 0 THEN EntryRemSec := 0; END_IF;
        MachineHomingInstruction := CONCAT('HX0 - Maintien homme-mort neutre: ',
                                           CONCAT(INT_TO_STRING(EntryRemSec), 's (secours: N2)'));
        MachineHomingActionText  := CONCAT('[HOMING] Maintenir HOMME-MORT neutre: ',
                                           CONCAT(INT_TO_STRING(EntryRemSec), 's'));
    ELSE
        EntryRemSec := DINT_TO_INT((TIME_TO_DINT(Cfg.CfgEntryHoldTime) + DINT#999) / DINT#1000);
        MachineHomingInstruction := CONCAT('HX0 - Tenir homme-mort ',
                                           CONCAT(INT_TO_STRING(EntryRemSec), 's neutre (ou N2)'));
        MachineHomingActionText  := '[HOMING] Tenir HOMME-MORT 5s NEUTRE pour lancer (ou N2)';
    END_IF;
ELSIF ModeIsMaint2 THEN
    MachineHomingStep := E_MachineHomingStep.BOTH_NOT_HOMED;
    IF NOT BootReady THEN
        MachineHomingInstruction := 'HX0 - Attente prets codeurs/boot (N2 libre)';
        MachineHomingActionText  := '[HOMING] Attente codeurs prets...';
    ELSIF EntryHoldTimer.ET >= T#1500ms THEN
        EntryRemSec := DINT_TO_INT((TIME_TO_DINT(Cfg.CfgEntryHoldTime - EntryHoldTimer.ET) + DINT#999) / DINT#1000);
        IF EntryRemSec < 0 THEN EntryRemSec := 0; END_IF;
        MachineHomingInstruction := CONCAT('HX0 - LANCEMENT HOMING DANS ',
                                           CONCAT(INT_TO_STRING(EntryRemSec), 's (lacher=annul.)'));
        MachineHomingActionText  := CONCAT('[HOMING] LANCEMENT DANS ',
                                           CONCAT(INT_TO_STRING(EntryRemSec), 's - LACHER POUR ANNULER'));
    ELSIF ProvisionalAborted THEN
        MachineHomingInstruction := 'HX0 - Altimetrie non calibree (N2 secours libre)';
        MachineHomingActionText  := '[HOMING] N2 libre - Homme-mort 5s neutre ou Start IHM';
    ELSE
        MachineHomingInstruction := 'HX0 - N2 libre actif | Homing: homme-mort 5s ou Start';
        MachineHomingActionText  := '[HOMING] N2 libre - Homme-mort 5s neutre ou Start IHM';
    END_IF;
ELSE
    MachineHomingStep := E_MachineHomingStep.BOTH_NOT_HOMED;
    IF ProvisionalAborted THEN
        MachineHomingInstruction := 'HX0 - Altimetrie non calibree: passer N1/N2';
        MachineHomingActionText  := '[HOMING] Non calibre - Passer en MAINT_N1 ou MAINT_N2';
    ELSE
        MachineHomingInstruction := 'HX0 - Non reference : passer en MAINT_N1 ou N2';
        MachineHomingActionText  := '[HOMING] Non reference - Passer en MAINT_N1 ou MAINT_N2';
    END_IF;
END_IF;

IF LatchedEdge.Q THEN
    MachineHomingStepAtError := MachineHomingStep;
END_IF;

Ready := Enable AND NOT Fault.Latched;
PrevMode := Mode;
FirstScanDone := TRUE;
{endregion}

          
END_FUNCTION_BLOCK

(* ======================================================================= 🧩 FB_FaultCore — Socle de remplissage de ST_Fault (vue live + vue latchée) ─────────────────────────────────────────────────────────────── 🎯 Rôle : à partir d'une LISTE de causes en clair (ARRAY[0..15] OF ST_FaultCause), produire la brique ST_Fault : • Error / ErrorId : vue LIVE, suit les causes Active, retombe seule. • Latched / LatchedId: vue LATCHÉE, chaque bit figé à l'apparition d'une cause `Active AND Latching`, conservé jusqu'au front Reset. 🔒 Sécurité : - interlock TOUJOURS sur `Causes[i].Active` (cause brute), jamais sur le latch. - Reset TOUJOURS effectif, jamais conditionné (std §9) — agit même Enable=FALSE. - Latching=FALSE → cause visible en LIVE seulement (fail-safe : reste visible). - un défaut laté non acquitté reste publié même FB désactivé (pas d'effacement silencieux sur bascule Enable OFF→ON sans Reset). - une cause à acquitter réapparue re-arme son bit (ré-alarme). 🧬 Un seul socle, réutilisé par tout FB `standard` qui expose un ST_Fault. Pas de State, pas de Warning, pas de texte — hors périmètre de ce socle. 📄 Doc : DOC/STDS/CODE_QUALITY_STANDARDS.md §2quinquies / §9 ======================================================================= *)
FUNCTION_BLOCK FB_FaultCore
  VAR_INPUT
    Enable : BOOL;  (* --> [CMD] Autorisation générale du FB porteur *)
    Reset : BOOL;  (* --> [CMD] Front d'acquittement (jamais conditionné, §9) *)
    Causes : ARRAY[0..15] OF ST_FaultCause;  (* --> [CMD] Liste des causes en clair (Active / Latching / Texte) *)
  END_VAR
  VAR_OUTPUT
    Ready : BOOL;  (* <-- [STAT] FB porteur autorisé (= Enable) *)
    Fault : ST_Fault;  (* <-- [DIAG] Brique défaut (mappée 1:1 sur la sortie du FB porteur) *)
  END_VAR
  VAR
    ResetEdge : R_TRIG;  (* . [LOC] Front montant Reset *)
    Latch : ARRAY[0..15] OF BOOL;  (* . [LOC] Bit laté par cause, jusqu'au Reset *)
    i : INT;  (* . [LOC] Index de parcours de la liste *)
  END_VAR

            

{region "§1 Reset (front, toujours effectif)"}
// Front Reset : efface tous les latches. Jamais conditionné, agit même Enable=FALSE (§9).
Ready := Enable;
ResetEdge(CLK := Reset);
IF ResetEdge.Q THEN
    FOR i := 0 TO 15 DO Latch[i] := FALSE; END_FOR;
END_IF;
{endregion}

{region "§2 Vue LIVE — Error / ErrorId"}
// Bitfield des causes présentes MAINTENANT. Retombe seule à 0 quand les causes disparaissent.
// Non évaluée si Enable=FALSE (pas de lecture de cause hors autorisation).
Fault.ErrorId := 0;
IF Enable THEN
    FOR i := 0 TO 15 DO
        IF Causes[i].Active THEN
            Fault.ErrorId := Fault.ErrorId OR SHL(WORD#1, INT_TO_DWORD(i));
        END_IF;
    END_FOR;
END_IF;
Fault.Error := (Fault.ErrorId <> 0);
{endregion}

{region "§3 Armement des latches (causes à acquitter)"}
// Une cause Active ET Latching arme son bit ; le bit reste jusqu'au front Reset (§1),
// même si la cause disparaît. Réapparition => ré-armement (ré-alarme).
IF Enable THEN
    FOR i := 0 TO 15 DO
        IF Causes[i].Active AND Causes[i].Latching THEN
            Latch[i] := TRUE;
        END_IF;
    END_FOR;
END_IF;
{endregion}

{region "§4 Vue LATCHÉE — Latched / LatchedId"}
// Toujours publiée, y compris Enable=FALSE : un défaut non acquitté reste visible.
Fault.LatchedId := 0;
FOR i := 0 TO 15 DO
    IF Latch[i] THEN
        Fault.LatchedId := Fault.LatchedId OR SHL(WORD#1, INT_TO_DWORD(i));
    END_IF;
END_FOR;
Fault.Latched := (Fault.LatchedId <> 0);
{endregion}

          
END_FUNCTION_BLOCK
